(* IEC 61131-3 sources: AXOpen/src/template.axolibrary/ctrl/src/TemplateComponent, 1 file *)

(* ---- TemplateComponent.st ---- *)
USING AXOpen.Core;
USING AXOpen.Messaging;
USING AXOpen.Messaging.Static;
USING AXOpen.Components.Abstractions;
USING Siemens.Simatic.Hardware.Utilities;

NAMESPACE Template.Axolibrary
    {S7.extern=ReadWrite}
    CLASS TemplateComponent EXTENDS AXOpen.Core.AxoComponent
        VAR PUBLIC // HEADER
            {#ix-attr:[ReadOnly()]}
            Progress       :   INT;
        END_VAR

        VAR PUBLIC // TASKS
            {#ix-attr:[Container(Layout.Wrap)]}
            {#ix-attr:[ComponentDetails("Tasks")]}
            {#ix-set:AttributeName = "<#Restore#>"}
            RestoreTask : AXOpen.Core.AxoTask;
        END_VAR

        VAR PUBLIC // TEMPLATE TASKS
            {#ix-attr:[Container(Layout.Wrap)]}
            {#ix-attr:[ComponentDetails("Template tasks")]}
            {#ix-set:AttributeName = "<#TemplateTask_10steps_1#>"}
            TemplateTask_10steps_1 : AXOpen.Core.AxoTask;
            {#ix-attr:[Container(Layout.Wrap)]}
            {#ix-attr:[ComponentDetails("Template tasks")]}
            {#ix-set:AttributeName = "<#TemplateTask_10steps_2#>"}
            TemplateTask_10steps_2 : AXOpen.Core.AxoTask;
            {#ix-attr:[Container(Layout.Wrap)]}
            {#ix-attr:[ComponentDetails("Template tasks")]}
            {#ix-set:AttributeName = "<#TemplateTask_10steps_3#>"}
            TemplateTask_10steps_3 : AXOpen.Core.AxoTask;
            {#ix-attr:[Container(Layout.Wrap)]}
            {#ix-attr:[ComponentDetails("Template tasks")]}
            {#ix-set:AttributeName = "<#TemplateTask_10steps_4#>"}
            TemplateTask_10steps_4 : AXOpen.Core.AxoTask;
            {#ix-attr:[Container(Layout.Wrap)]}
            {#ix-attr:[ComponentDetails("Template tasks")]}
            {#ix-set:AttributeName = "<#TemplateTask_10steps_5#>"}
            TemplateTask_10steps_5 : AXOpen.Core.AxoTask;
            {#ix-attr:[Container(Layout.Wrap)]}
            {#ix-attr:[ComponentDetails("Template tasks")]}
            {#ix-set:AttributeName = "<#TemplateTask_10steps_6#>"}
            TemplateTask_10steps_6 : AXOpen.Core.AxoTask;

            {#ix-attr:[Container(Layout.Wrap)]}
            {#ix-attr:[ComponentDetails("Template tasks")]}
            {#ix-set:AttributeName = "<#TemplateTask_20steps_1#>"}
            TemplateTask_20steps_1 : AXOpen.Core.AxoTask;
            {#ix-attr:[Container(Layout.Wrap)]}
            {#ix-attr:[ComponentDetails("Template tasks")]}
            {#ix-set:AttributeName = "<#TemplateTask_20steps_2#>"}
            TemplateTask_20steps_2 : AXOpen.Core.AxoTask;
            {#ix-attr:[Container(Layout.Wrap)]}
            {#ix-attr:[ComponentDetails("Template tasks")]}
            {#ix-set:AttributeName = "<#TemplateTask_20steps_3#>"}
            TemplateTask_20steps_3 : AXOpen.Core.AxoTask;
            {#ix-attr:[Container(Layout.Wrap)]}
            {#ix-attr:[ComponentDetails("Template tasks")]}
            {#ix-set:AttributeName = "<#TemplateTask_20steps_4#>"}
            TemplateTask_20steps_4 : AXOpen.Core.AxoTask;
            {#ix-attr:[Container(Layout.Wrap)]}
            {#ix-attr:[ComponentDetails("Template tasks")]}
            {#ix-set:AttributeName = "<#TemplateTask_20steps_5#>"}
            TemplateTask_20steps_5 : AXOpen.Core.AxoTask;
            {#ix-attr:[Container(Layout.Wrap)]}
            {#ix-attr:[ComponentDetails("Template tasks")]}
            {#ix-set:AttributeName = "<#TemplateTask_20steps_6#>"}
            TemplateTask_20steps_6 : AXOpen.Core.AxoTask;

        END_VAR

        VAR PUBLIC // CONFIG
            {#ix-attr:[Container(Layout.Stack)]}
            {#ix-attr:[ComponentDetails("Config")]}
            {#ix-attr:[ReadOnly()]}
            Config  :   TemplateComponent_Config;
        END_VAR

        VAR PUBLIC // STATUS
            {#ix-attr:[Container(Layout.Stack)]}
            {#ix-attr:[ComponentDetails("Status")]}
            {#ix-attr:[ReadOnly()]}
            Status              :   TemplateComponent_Component_Status;
            Messenger           :   AXOpen.Messaging.Static.AxoMessenger;
            TaskMessenger       :   AXOpen.Messaging.Static.AxoMessenger;
        END_VAR

        VAR PUBLIC // HARDWARE SIGNALS
            {#ix-attr:[ComponentDetails("HARDWARE SIGNALS")]}
            {#ix-attr:[Container(Layout.Wrap)]}
            {#ix-attr:[Group(GroupLayout.GroupBox)]}
            {#ix-set:AttributeName = "<#Inputs#>"}
            {#ix-attr:[ReadOnly()]}
            Inputs              :  TemplateComponent_In;
            {#ix-attr:[ComponentDetails("HARDWARE SIGNALS")]}
            {#ix-attr:[Container(Layout.Wrap)]}
            {#ix-attr:[Group(GroupLayout.GroupBox)]}
            {#ix-set:AttributeName = "<#Outputs#>"}
            {#ix-attr:[ReadOnly()]}
            Outputs              :   TemplateComponent_Out;
        END_VAR

        VAR PUBLIC // HARDWARE DIAGNOSTICS TASK
            {#ix-attr:[Container(Layout.Stack)]}
            {#ix-attr:[ComponentDetails("Hardware diagnostics")]}
            {#ix-set:AttributeName = "<#Update diagnostics#>"}
            HardwareDiagnosticsTask :   AXOpen.Io.AxoHardwareDiagnostics;
        END_VAR

        VAR PRIVATE
            _progress       :   INT;
            _infoTimer      :   AXOpen.Timers.OnDelayTimer;
            _errorTimer     :   AXOpen.Timers.OnDelayTimer;
            _data_in        :   ARRAY[0..254] OF BYTE;
            _data_out_1     :   ARRAY[0..0] OF BYTE;
            _data_out_2     :   ARRAY[0..1] OF BYTE;
            _data_out_4     :   ARRAY[0..3] OF BYTE;
            _data_out_8     :   ARRAY[0..7] OF BYTE;
            _data_out_255   :   ARRAY[0..254] OF BYTE;
            _word           :   WORD;
            _dword          :   DWORD;

            _initHwCheckDone        :   BOOL;
            _retval                 :   WORD;
            _geoAddr                :   GeoAddr;
            _outHwid                :   UINT;
            _blink                  :   AXOpen.Timers.AxoBlinker;
            _inputsAddress          :   UDINT;
            _inputsCount            :   UINT;
            _outputsAddress         :   UDINT;
            _outputsCount           :   UINT;
        END_VAR

        ///<summary>
        /// Runs tasks and logic of this component.
        /// >[!IMPORTANT] This method must or one of its overloads be called cyclically.
        ///</summary>
        METHOD PUBLIC Run
            VAR_INPUT
                inParent    :   IAxoObject;
                hwID        :   UINT;
            END_VAR

            SUPER.Run(inParent);

            Messenger.Serve(THIS);

            Progress := _progress;

            IF NOT _initHwCheckDone THEN
                IF inParent = NULL THEN
                    Messenger.Activate(UINT#700, eAxoMessageCategory#ProgrammingError);
                    Status.Error.Id := UINT#700;
                    RETURN;
                END_IF;
                IF hwID = UINT#0 THEN
                    Messenger.Activate(UINT#701, eAxoMessageCategory#ProgrammingError);
                    Status.Error.Id := UINT#701;
                    RETURN;
                END_IF;

                Config.HWIDs.HW_Device := hwID;
                _retval := ReadSlotFromHardwareID(hardwareID := Config.HWIDs.HW_Device, geoAddr :=_geoAddr);
                IF _retval = WORD#8090 THEN
                    Messenger.Activate(UINT#702,eAxoMessageCategory#Error);
                    Status.Error.Id := UINT#702;
                    RETURN;
                END_IF;

                //******************Slot 1*****************//
                _geoAddr.Slot   :=  UINT#1;
                _geoAddr.HardwareType := UINT#4; // (4-Module)
                _retval := ReadHardwareIDFromSlot(geoAddr := _geoAddr, hardwareID => Config.HWIDs.HwID_in_1);
                IF Config.HWIDs.HwID_in_1 = UINT#0 THEN
                    Messenger.Activate(UINT#710,eAxoMessageCategory#Error);
                    Status.Error.Id := UINT#710;
                    RETURN;
                END_IF;
                IF _retval = WORD#8091 THEN
                    Messenger.Activate(UINT#711,eAxoMessageCategory#Error);
                    Status.Error.Id := UINT#711;
                    RETURN;
                END_IF;
                IF _retval = WORD#8094 THEN
                    Messenger.Activate(UINT#712,eAxoMessageCategory#Error);
                    Status.Error.Id := UINT#712;
                    RETURN;
                END_IF;
                IF _retval = WORD#8095 THEN
                    Messenger.Activate(UINT#713,eAxoMessageCategory#Error);
                    Status.Error.Id := UINT#713;
                    RETURN;
                END_IF;
                IF _retval = WORD#8096 THEN
                    Messenger.Activate(UINT#714,eAxoMessageCategory#Error);
                    Status.Error.Id := UINT#714;
                    RETURN;
                END_IF;
                IF _retval = WORD#8097 THEN
                    Messenger.Activate(UINT#715,eAxoMessageCategory#Error);
                    Status.Error.Id := UINT#715;
                    RETURN;
                END_IF;
                ReadHardwareIOAddress(hardwareID := (Config.HWIDs.HwID_in_1) , inputStartAddress => _inputsAddress , inputCount => _inputsCount , outputStartAddress => _outputsAddress , outputCount => _outputsCount);
                IF _inputsCount <> UINT#8 OR _outputsCount <> UINT#0 THEN
                    Messenger.Activate(UINT#716,eAxoMessageCategory#Error);
                    Status.Error.Id := UINT#716;
                    RETURN;
                END_IF;
                //******************Slot 2*****************//
                _geoAddr.Slot   :=  UINT#2;
                _geoAddr.HardwareType := UINT#4; // (4-Module)
                _retval := ReadHardwareIDFromSlot(geoAddr := _geoAddr, hardwareID => Config.HWIDs.HwID_in_2);
                IF Config.HWIDs.HwID_in_2 = UINT#0 THEN
                    Messenger.Activate(UINT#720,eAxoMessageCategory#Error);
                    Status.Error.Id := UINT#720;
                    RETURN;
                END_IF;
                IF _retval = WORD#8091 THEN
                    Messenger.Activate(UINT#721,eAxoMessageCategory#Error);
                    Status.Error.Id := UINT#721;
                    RETURN;
                END_IF;
                IF _retval = WORD#8094 THEN
                    Messenger.Activate(UINT#722,eAxoMessageCategory#Error);
                    Status.Error.Id := UINT#722;
                    RETURN;
                END_IF;
                IF _retval = WORD#8095 THEN
                    Messenger.Activate(UINT#723,eAxoMessageCategory#Error);
                    Status.Error.Id := UINT#723;
                    RETURN;
                END_IF;
                IF _retval = WORD#8096 THEN
                    Messenger.Activate(UINT#724,eAxoMessageCategory#Error);
                    Status.Error.Id := UINT#724;
                    RETURN;
                END_IF;
                IF _retval = WORD#8097 THEN
                    Messenger.Activate(UINT#725,eAxoMessageCategory#Error);
                    Status.Error.Id := UINT#725;
                    RETURN;
                END_IF;
                ReadHardwareIOAddress(hardwareID := (Config.HWIDs.HwID_in_2) , inputStartAddress => _inputsAddress , inputCount => _inputsCount , outputStartAddress => _outputsAddress , outputCount => _outputsCount);
                IF _inputsCount <> UINT#8 OR _outputsCount <> UINT#0 THEN
                    Messenger.Activate(UINT#726,eAxoMessageCategory#Error);
                    Status.Error.Id := UINT#726;
                    RETURN;
                END_IF;
                //******************Slot 3*****************//
                _geoAddr.Slot   :=  UINT#3;
                _geoAddr.HardwareType := UINT#4; // (4-Module)
                _retval := ReadHardwareIDFromSlot(geoAddr := _geoAddr, hardwareID => Config.HWIDs.HwID_in_3);
                IF Config.HWIDs.HwID_in_1 = UINT#0 THEN
                    Messenger.Activate(UINT#730,eAxoMessageCategory#Error);
                    Status.Error.Id := UINT#730;
                    RETURN;
                END_IF;
                IF _retval = WORD#8091 THEN
                    Messenger.Activate(UINT#731,eAxoMessageCategory#Error);
                    Status.Error.Id := UINT#731;
                    RETURN;
                END_IF;
                IF _retval = WORD#8094 THEN
                    Messenger.Activate(UINT#732,eAxoMessageCategory#Error);
                    Status.Error.Id := UINT#732;
                    RETURN;
                END_IF;
                IF _retval = WORD#8095 THEN
                    Messenger.Activate(UINT#733,eAxoMessageCategory#Error);
                    Status.Error.Id := UINT#733;
                    RETURN;
                END_IF;
                IF _retval = WORD#8096 THEN
                    Messenger.Activate(UINT#734,eAxoMessageCategory#Error);
                    Status.Error.Id := UINT#734;
                    RETURN;
                END_IF;
                IF _retval = WORD#8097 THEN
                    Messenger.Activate(UINT#735,eAxoMessageCategory#Error);
                    Status.Error.Id := UINT#735;
                    RETURN;
                END_IF;
                ReadHardwareIOAddress(hardwareID := (Config.HWIDs.HwID_in_3) , inputStartAddress => _inputsAddress , inputCount => _inputsCount , outputStartAddress => _outputsAddress , outputCount => _outputsCount);
                IF _inputsCount <> UINT#8 OR _outputsCount <> UINT#0 THEN
                    Messenger.Activate(UINT#736,eAxoMessageCategory#Error);
                    Status.Error.Id := UINT#736;
                    RETURN;
                END_IF;
                //******************Slot 4*****************//
                _geoAddr.Slot   :=  UINT#4;
                _geoAddr.HardwareType := UINT#4; // (4-Module)
                _retval := ReadHardwareIDFromSlot(geoAddr := _geoAddr, hardwareID => Config.HWIDs.HwID_in_4);
                IF Config.HWIDs.HwID_in_4 = UINT#0 THEN
                    Messenger.Activate(UINT#740,eAxoMessageCategory#Error);
                    Status.Error.Id := UINT#740;
                    RETURN;
                END_IF;
                IF _retval = WORD#8091 THEN
                    Messenger.Activate(UINT#741,eAxoMessageCategory#Error);
                    Status.Error.Id := UINT#741;
                    RETURN;
                END_IF;
                IF _retval = WORD#8094 THEN
                    Messenger.Activate(UINT#742,eAxoMessageCategory#Error);
                    Status.Error.Id := UINT#742;
                    RETURN;
                END_IF;
                IF _retval = WORD#8095 THEN
                    Messenger.Activate(UINT#743,eAxoMessageCategory#Error);
                    Status.Error.Id := UINT#743;
                    RETURN;
                END_IF;
                IF _retval = WORD#8096 THEN
                    Messenger.Activate(UINT#744,eAxoMessageCategory#Error);
                    Status.Error.Id := UINT#744;
                    RETURN;
                END_IF;
                IF _retval = WORD#8097 THEN
                    Messenger.Activate(UINT#745,eAxoMessageCategory#Error);
                    Status.Error.Id := UINT#745;
                    RETURN;
                END_IF;
                ReadHardwareIOAddress(hardwareID := (Config.HWIDs.HwID_in_4) , inputStartAddress => _inputsAddress , inputCount => _inputsCount , outputStartAddress => _outputsAddress , outputCount => _outputsCount);
                IF _inputsCount <> UINT#8 OR _outputsCount <> UINT#0 THEN
                    Messenger.Activate(UINT#746,eAxoMessageCategory#Error);
                    Status.Error.Id := UINT#746;
                    RETURN;
                END_IF;
                //******************Slot 5*****************//
                _geoAddr.Slot   :=  UINT#5;
                _geoAddr.HardwareType := UINT#4; // (4-Module)
                _retval := ReadHardwareIDFromSlot(geoAddr := _geoAddr, hardwareID => Config.HWIDs.HwID_in_5);
                IF Config.HWIDs.HwID_in_5 = UINT#0 THEN
                    Messenger.Activate(UINT#750,eAxoMessageCategory#Error);
                    Status.Error.Id := UINT#750;
                    RETURN;
                END_IF;
                IF _retval = WORD#8091 THEN
                    Messenger.Activate(UINT#751,eAxoMessageCategory#Error);
                    Status.Error.Id := UINT#751;
                    RETURN;
                END_IF;
                IF _retval = WORD#8094 THEN
                    Messenger.Activate(UINT#752,eAxoMessageCategory#Error);
                    Status.Error.Id := UINT#752;
                    RETURN;
                END_IF;
                IF _retval = WORD#8095 THEN
                    Messenger.Activate(UINT#753,eAxoMessageCategory#Error);
                    Status.Error.Id := UINT#753;
                    RETURN;
                END_IF;
                IF _retval = WORD#8096 THEN
                    Messenger.Activate(UINT#754,eAxoMessageCategory#Error);
                    Status.Error.Id := UINT#754;
                    RETURN;
                END_IF;
                IF _retval = WORD#8097 THEN
                    Messenger.Activate(UINT#755,eAxoMessageCategory#Error);
                    Status.Error.Id := UINT#755;
                    RETURN;
                END_IF;
                ReadHardwareIOAddress(hardwareID := (Config.HWIDs.HwID_in_5) , inputStartAddress => _inputsAddress , inputCount => _inputsCount , outputStartAddress => _outputsAddress , outputCount => _outputsCount);
                IF _inputsCount <> UINT#8 OR _outputsCount <> UINT#0 THEN
                    Messenger.Activate(UINT#756,eAxoMessageCategory#Error);
                    Status.Error.Id := UINT#756;
                    RETURN;
                END_IF;
                //******************Slot 6*****************//
                _geoAddr.Slot   :=  UINT#6;
                _geoAddr.HardwareType := UINT#4; // (4-Module)
                _retval := ReadHardwareIDFromSlot(geoAddr := _geoAddr, hardwareID => Config.HWIDs.HwID_in_6);
                IF Config.HWIDs.HwID_in_6 = UINT#0 THEN
                    Messenger.Activate(UINT#760,eAxoMessageCategory#Error);
                    Status.Error.Id := UINT#760;
                    RETURN;
                END_IF;
                IF _retval = WORD#8091 THEN
                    Messenger.Activate(UINT#761,eAxoMessageCategory#Error);
                    Status.Error.Id := UINT#761;
                    RETURN;
                END_IF;
                IF _retval = WORD#8094 THEN
                    Messenger.Activate(UINT#762,eAxoMessageCategory#Error);
                    Status.Error.Id := UINT#762;
                    RETURN;
                END_IF;
                IF _retval = WORD#8095 THEN
                    Messenger.Activate(UINT#763,eAxoMessageCategory#Error);
                    Status.Error.Id := UINT#763;
                    RETURN;
                END_IF;
                IF _retval = WORD#8096 THEN
                    Messenger.Activate(UINT#764,eAxoMessageCategory#Error);
                    Status.Error.Id := UINT#764;
                    RETURN;
                END_IF;
                IF _retval = WORD#8097 THEN
                    Messenger.Activate(UINT#765,eAxoMessageCategory#Error);
                    Status.Error.Id := UINT#765;
                    RETURN;
                END_IF;
                ReadHardwareIOAddress(hardwareID := (Config.HWIDs.HwID_in_6) , inputStartAddress => _inputsAddress , inputCount => _inputsCount , outputStartAddress => _outputsAddress , outputCount => _outputsCount);
                IF _inputsCount <> UINT#8 OR _outputsCount <> UINT#0 THEN
                    Messenger.Activate(UINT#766,eAxoMessageCategory#Error);
                    Status.Error.Id := UINT#766;
                    RETURN;
                END_IF;
                //******************Slot 7*****************//
                _geoAddr.Slot   :=  UINT#7;
                _geoAddr.HardwareType := UINT#4; // (4-Module)
                _retval := ReadHardwareIDFromSlot(geoAddr := _geoAddr, hardwareID => Config.HWIDs.HwID_in_7);
                IF Config.HWIDs.HwID_in_7 = UINT#0 THEN
                    Messenger.Activate(UINT#770,eAxoMessageCategory#Error);
                    Status.Error.Id := UINT#770;
                    RETURN;
                END_IF;
                IF _retval = WORD#8091 THEN
                    Messenger.Activate(UINT#771,eAxoMessageCategory#Error);
                    Status.Error.Id := UINT#771;
                    RETURN;
                END_IF;
                IF _retval = WORD#8094 THEN
                    Messenger.Activate(UINT#772,eAxoMessageCategory#Error);
                    Status.Error.Id := UINT#772;
                    RETURN;
                END_IF;
                IF _retval = WORD#8095 THEN
                    Messenger.Activate(UINT#773,eAxoMessageCategory#Error);
                    Status.Error.Id := UINT#773;
                    RETURN;
                END_IF;
                IF _retval = WORD#8096 THEN
                    Messenger.Activate(UINT#774,eAxoMessageCategory#Error);
                    Status.Error.Id := UINT#774;
                    RETURN;
                END_IF;
                IF _retval = WORD#8097 THEN
                    Messenger.Activate(UINT#775,eAxoMessageCategory#Error);
                    Status.Error.Id := UINT#775;
                    RETURN;
                END_IF;
                ReadHardwareIOAddress(hardwareID := (Config.HWIDs.HwID_in_7) , inputStartAddress => _inputsAddress , inputCount => _inputsCount , outputStartAddress => _outputsAddress , outputCount => _outputsCount);
                IF _inputsCount <> UINT#8 OR _outputsCount <> UINT#0 THEN
                    Messenger.Activate(UINT#776,eAxoMessageCategory#Error);
                    Status.Error.Id := UINT#776;
                    RETURN;
                END_IF;
                //******************Slot 8*****************//
                _geoAddr.Slot   :=  UINT#8;
                _geoAddr.HardwareType := UINT#4; // (4-Module)
                _retval := ReadHardwareIDFromSlot(geoAddr := _geoAddr, hardwareID => Config.HWIDs.HwID_in_8);
                IF Config.HWIDs.HwID_in_8 = UINT#0 THEN
                    Messenger.Activate(UINT#780,eAxoMessageCategory#Error);
                    Status.Error.Id := UINT#780;
                    RETURN;
                END_IF;
                IF _retval = WORD#8091 THEN
                    Messenger.Activate(UINT#781,eAxoMessageCategory#Error);
                    Status.Error.Id := UINT#781;
                    RETURN;
                END_IF;
                IF _retval = WORD#8094 THEN
                    Messenger.Activate(UINT#782,eAxoMessageCategory#Error);
                    Status.Error.Id := UINT#782;
                    RETURN;
                END_IF;
                IF _retval = WORD#8095 THEN
                    Messenger.Activate(UINT#783,eAxoMessageCategory#Error);
                    Status.Error.Id := UINT#783;
                    RETURN;
                END_IF;
                IF _retval = WORD#8096 THEN
                    Messenger.Activate(UINT#784,eAxoMessageCategory#Error);
                    Status.Error.Id := UINT#784;
                    RETURN;
                END_IF;
                IF _retval = WORD#8097 THEN
                    Messenger.Activate(UINT#785,eAxoMessageCategory#Error);
                    Status.Error.Id := UINT#785;
                    RETURN;
                END_IF;
                ReadHardwareIOAddress(hardwareID := (Config.HWIDs.HwID_in_8) , inputStartAddress => _inputsAddress , inputCount => _inputsCount , outputStartAddress => _outputsAddress , outputCount => _outputsCount);
                IF _inputsCount <> UINT#8 OR _outputsCount <> UINT#0 THEN
                    Messenger.Activate(UINT#786,eAxoMessageCategory#Error);
                    Status.Error.Id := UINT#786;
                    RETURN;
                END_IF;
                //******************Slot 9*****************//
                _geoAddr.Slot   :=  UINT#9;
                _geoAddr.HardwareType := UINT#4; // (4-Module)
                _retval := ReadHardwareIDFromSlot(geoAddr := _geoAddr, hardwareID => Config.HWIDs.HwID_in_9);
                IF Config.HWIDs.HwID_in_9 = UINT#0 THEN
                    Messenger.Activate(UINT#790,eAxoMessageCategory#Error);
                    Status.Error.Id := UINT#790;
                    RETURN;
                END_IF;
                IF _retval = WORD#8091 THEN
                    Messenger.Activate(UINT#791,eAxoMessageCategory#Error);
                    Status.Error.Id := UINT#791;
                    RETURN;
                END_IF;
                IF _retval = WORD#8094 THEN
                    Messenger.Activate(UINT#792,eAxoMessageCategory#Error);
                    Status.Error.Id := UINT#792;
                    RETURN;
                END_IF;
                IF _retval = WORD#8095 THEN
                    Messenger.Activate(UINT#793,eAxoMessageCategory#Error);
                    Status.Error.Id := UINT#793;
                    RETURN;
                END_IF;
                IF _retval = WORD#8096 THEN
                    Messenger.Activate(UINT#794,eAxoMessageCategory#Error);
                    Status.Error.Id := UINT#794;
                    RETURN;
                END_IF;
                IF _retval = WORD#8097 THEN
                    Messenger.Activate(UINT#795,eAxoMessageCategory#Error);
                    Status.Error.Id := UINT#795;
                    RETURN;
                END_IF;
                ReadHardwareIOAddress(hardwareID := (Config.HWIDs.HwID_in_9) , inputStartAddress => _inputsAddress , inputCount => _inputsCount , outputStartAddress => _outputsAddress , outputCount => _outputsCount);
                IF _inputsCount <> UINT#8 OR _outputsCount <> UINT#0 THEN
                    Messenger.Activate(UINT#796,eAxoMessageCategory#Error);
                    Status.Error.Id := UINT#796;
                    RETURN;
                END_IF;
                //******************Slot 10*****************//
                _geoAddr.Slot   :=  UINT#10;
                _geoAddr.HardwareType := UINT#4; // (4-Module)
                _retval := ReadHardwareIDFromSlot(geoAddr := _geoAddr, hardwareID => Config.HWIDs.HwID_in_10);
                IF Config.HWIDs.HwID_in_10 = UINT#0 THEN
                    Messenger.Activate(UINT#800,eAxoMessageCategory#Error);
                    Status.Error.Id := UINT#800;
                    RETURN;
                END_IF;
                IF _retval = WORD#8091 THEN
                    Messenger.Activate(UINT#801,eAxoMessageCategory#Error);
                    Status.Error.Id := UINT#801;
                    RETURN;
                END_IF;
                IF _retval = WORD#8094 THEN
                    Messenger.Activate(UINT#802,eAxoMessageCategory#Error);
                    Status.Error.Id := UINT#802;
                    RETURN;
                END_IF;
                IF _retval = WORD#8095 THEN
                    Messenger.Activate(UINT#803,eAxoMessageCategory#Error);
                    Status.Error.Id := UINT#803;
                    RETURN;
                END_IF;
                IF _retval = WORD#8096 THEN
                    Messenger.Activate(UINT#804,eAxoMessageCategory#Error);
                    Status.Error.Id := UINT#804;
                    RETURN;
                END_IF;
                IF _retval = WORD#8097 THEN
                    Messenger.Activate(UINT#805,eAxoMessageCategory#Error);
                    Status.Error.Id := UINT#805;
                    RETURN;
                END_IF;
                ReadHardwareIOAddress(hardwareID := (Config.HWIDs.HwID_in_10) , inputStartAddress => _inputsAddress , inputCount => _inputsCount , outputStartAddress => _outputsAddress , outputCount => _outputsCount);
                IF _inputsCount <> UINT#8 OR _outputsCount <> UINT#0 THEN
                    Messenger.Activate(UINT#806,eAxoMessageCategory#Error);
                    Status.Error.Id := UINT#806;
                    RETURN;
                END_IF;
                //******************Slot 11*****************//
                _geoAddr.Slot   :=  UINT#11;
                _geoAddr.HardwareType := UINT#4; // (4-Module)
                _retval := ReadHardwareIDFromSlot(geoAddr := _geoAddr, hardwareID => Config.HWIDs.HwID_in_11);
                IF Config.HWIDs.HwID_in_11 = UINT#0 THEN
                    Messenger.Activate(UINT#810,eAxoMessageCategory#Error);
                    Status.Error.Id := UINT#810;
                    RETURN;
                END_IF;
                IF _retval = WORD#8091 THEN
                    Messenger.Activate(UINT#811,eAxoMessageCategory#Error);
                    Status.Error.Id := UINT#811;
                    RETURN;
                END_IF;
                IF _retval = WORD#8094 THEN
                    Messenger.Activate(UINT#812,eAxoMessageCategory#Error);
                    Status.Error.Id := UINT#812;
                    RETURN;
                END_IF;
                IF _retval = WORD#8095 THEN
                    Messenger.Activate(UINT#813,eAxoMessageCategory#Error);
                    Status.Error.Id := UINT#813;
                    RETURN;
                END_IF;
                IF _retval = WORD#8096 THEN
                    Messenger.Activate(UINT#814,eAxoMessageCategory#Error);
                    Status.Error.Id := UINT#814;
                    RETURN;
                END_IF;
                IF _retval = WORD#8097 THEN
                    Messenger.Activate(UINT#815,eAxoMessageCategory#Error);
                    Status.Error.Id := UINT#815;
                    RETURN;
                END_IF;
                ReadHardwareIOAddress(hardwareID := (Config.HWIDs.HwID_in_11) , inputStartAddress => _inputsAddress , inputCount => _inputsCount , outputStartAddress => _outputsAddress , outputCount => _outputsCount);
                IF _inputsCount <> UINT#8 OR _outputsCount <> UINT#0 THEN
                    Messenger.Activate(UINT#816,eAxoMessageCategory#Error);
                    Status.Error.Id := UINT#816;
                    RETURN;
                END_IF;
                //******************Slot 12*****************//
                _geoAddr.Slot   :=  UINT#12;
                _geoAddr.HardwareType := UINT#4; // (4-Module)
                _retval := ReadHardwareIDFromSlot(geoAddr := _geoAddr, hardwareID => Config.HWIDs.HwID_in_12);
                IF Config.HWIDs.HwID_in_12 = UINT#0 THEN
                    Messenger.Activate(UINT#820,eAxoMessageCategory#Error);
                    Status.Error.Id := UINT#820;
                    RETURN;
                END_IF;
                IF _retval = WORD#8091 THEN
                    Messenger.Activate(UINT#821,eAxoMessageCategory#Error);
                    Status.Error.Id := UINT#821;
                    RETURN;
                END_IF;
                IF _retval = WORD#8094 THEN
                    Messenger.Activate(UINT#822,eAxoMessageCategory#Error);
                    Status.Error.Id := UINT#822;
                    RETURN;
                END_IF;
                IF _retval = WORD#8095 THEN
                    Messenger.Activate(UINT#823,eAxoMessageCategory#Error);
                    Status.Error.Id := UINT#823;
                    RETURN;
                END_IF;
                IF _retval = WORD#8096 THEN
                    Messenger.Activate(UINT#824,eAxoMessageCategory#Error);
                    Status.Error.Id := UINT#824;
                    RETURN;
                END_IF;
                IF _retval = WORD#8097 THEN
                    Messenger.Activate(UINT#825,eAxoMessageCategory#Error);
                    Status.Error.Id := UINT#825;
                    RETURN;
                END_IF;
                ReadHardwareIOAddress(hardwareID := (Config.HWIDs.HwID_in_12) , inputStartAddress => _inputsAddress , inputCount => _inputsCount , outputStartAddress => _outputsAddress , outputCount => _outputsCount);
                IF _inputsCount <> UINT#8 OR _outputsCount <> UINT#0 THEN
                    Messenger.Activate(UINT#826,eAxoMessageCategory#Error);
                    Status.Error.Id := UINT#826;
                    RETURN;
                END_IF;
                //******************Slot 13*****************//
                _geoAddr.Slot   :=  UINT#13;
                _geoAddr.HardwareType := UINT#4; // (4-Module)
                _retval := ReadHardwareIDFromSlot(geoAddr := _geoAddr, hardwareID => Config.HWIDs.HwID_in_13);
                IF Config.HWIDs.HwID_in_13 = UINT#0 THEN
                    Messenger.Activate(UINT#830,eAxoMessageCategory#Error);
                    Status.Error.Id := UINT#830;
                    RETURN;
                END_IF;
                IF _retval = WORD#8091 THEN
                    Messenger.Activate(UINT#831,eAxoMessageCategory#Error);
                    Status.Error.Id := UINT#831;
                    RETURN;
                END_IF;
                IF _retval = WORD#8094 THEN
                    Messenger.Activate(UINT#832,eAxoMessageCategory#Error);
                    Status.Error.Id := UINT#832;
                    RETURN;
                END_IF;
                IF _retval = WORD#8095 THEN
                    Messenger.Activate(UINT#833,eAxoMessageCategory#Error);
                    Status.Error.Id := UINT#833;
                    RETURN;
                END_IF;
                IF _retval = WORD#8096 THEN
                    Messenger.Activate(UINT#834,eAxoMessageCategory#Error);
                    Status.Error.Id := UINT#834;
                    RETURN;
                END_IF;
                IF _retval = WORD#8097 THEN
                    Messenger.Activate(UINT#835,eAxoMessageCategory#Error);
                    Status.Error.Id := UINT#835;
                    RETURN;
                END_IF;
                ReadHardwareIOAddress(hardwareID := (Config.HWIDs.HwID_in_13) , inputStartAddress => _inputsAddress , inputCount => _inputsCount , outputStartAddress => _outputsAddress , outputCount => _outputsCount);
                IF _inputsCount <> UINT#8 OR _outputsCount <> UINT#0 THEN
                    Messenger.Activate(UINT#836,eAxoMessageCategory#Error);
                    Status.Error.Id := UINT#836;
                    RETURN;
                END_IF;
                //******************Slot 14*****************//
                _geoAddr.Slot   :=  UINT#14;
                _geoAddr.HardwareType := UINT#4; // (4-Module)
                _retval := ReadHardwareIDFromSlot(geoAddr := _geoAddr, hardwareID => Config.HWIDs.HwID_in_14);
                IF Config.HWIDs.HwID_in_14 = UINT#0 THEN
                    Messenger.Activate(UINT#840,eAxoMessageCategory#Error);
                    Status.Error.Id := UINT#840;
                    RETURN;
                END_IF;
                IF _retval = WORD#8091 THEN
                    Messenger.Activate(UINT#841,eAxoMessageCategory#Error);
                    Status.Error.Id := UINT#841;
                    RETURN;
                END_IF;
                IF _retval = WORD#8094 THEN
                    Messenger.Activate(UINT#842,eAxoMessageCategory#Error);
                    Status.Error.Id := UINT#842;
                    RETURN;
                END_IF;
                IF _retval = WORD#8095 THEN
                    Messenger.Activate(UINT#843,eAxoMessageCategory#Error);
                    Status.Error.Id := UINT#843;
                    RETURN;
                END_IF;
                IF _retval = WORD#8096 THEN
                    Messenger.Activate(UINT#844,eAxoMessageCategory#Error);
                    Status.Error.Id := UINT#844;
                    RETURN;
                END_IF;
                IF _retval = WORD#8097 THEN
                    Messenger.Activate(UINT#845,eAxoMessageCategory#Error);
                    Status.Error.Id := UINT#845;
                    RETURN;
                END_IF;
                ReadHardwareIOAddress(hardwareID := (Config.HWIDs.HwID_in_14) , inputStartAddress => _inputsAddress , inputCount => _inputsCount , outputStartAddress => _outputsAddress , outputCount => _outputsCount);
                IF _inputsCount <> UINT#8 OR _outputsCount <> UINT#0 THEN
                    Messenger.Activate(UINT#846,eAxoMessageCategory#Error);
                    Status.Error.Id := UINT#846;
                    RETURN;
                END_IF;
                //******************Slot 15*****************//
                _geoAddr.Slot   :=  UINT#15;
                _geoAddr.HardwareType := UINT#4; // (4-Module)
                _retval := ReadHardwareIDFromSlot(geoAddr := _geoAddr, hardwareID => Config.HWIDs.HwID_in_15);
                IF Config.HWIDs.HwID_in_15 = UINT#0 THEN
                    Messenger.Activate(UINT#850,eAxoMessageCategory#Error);
                    Status.Error.Id := UINT#850;
                    RETURN;
                END_IF;
                IF _retval = WORD#8091 THEN
                    Messenger.Activate(UINT#851,eAxoMessageCategory#Error);
                    Status.Error.Id := UINT#851;
                    RETURN;
                END_IF;
                IF _retval = WORD#8094 THEN
                    Messenger.Activate(UINT#852,eAxoMessageCategory#Error);
                    Status.Error.Id := UINT#852;
                    RETURN;
                END_IF;
                IF _retval = WORD#8095 THEN
                    Messenger.Activate(UINT#853,eAxoMessageCategory#Error);
                    Status.Error.Id := UINT#853;
                    RETURN;
                END_IF;
                IF _retval = WORD#8096 THEN
                    Messenger.Activate(UINT#854,eAxoMessageCategory#Error);
                    Status.Error.Id := UINT#854;
                    RETURN;
                END_IF;
                IF _retval = WORD#8097 THEN
                    Messenger.Activate(UINT#855,eAxoMessageCategory#Error);
                    Status.Error.Id := UINT#855;
                    RETURN;
                END_IF;
                ReadHardwareIOAddress(hardwareID := (Config.HWIDs.HwID_in_15) , inputStartAddress => _inputsAddress , inputCount => _inputsCount , outputStartAddress => _outputsAddress , outputCount => _outputsCount);
                IF _inputsCount <> UINT#8 OR _outputsCount <> UINT#0 THEN
                    Messenger.Activate(UINT#856,eAxoMessageCategory#Error);
                    Status.Error.Id := UINT#856;
                    RETURN;
                END_IF;
                //******************Slot 16*****************//
                _geoAddr.Slot   :=  UINT#16;
                _geoAddr.HardwareType := UINT#4; // (4-Module)
                _retval := ReadHardwareIDFromSlot(geoAddr := _geoAddr, hardwareID => Config.HWIDs.HwID_in_16);
                IF Config.HWIDs.HwID_in_16 = UINT#0 THEN
                    Messenger.Activate(UINT#860,eAxoMessageCategory#Error);
                    Status.Error.Id := UINT#860;
                    RETURN;
                END_IF;
                IF _retval = WORD#8091 THEN
                    Messenger.Activate(UINT#861,eAxoMessageCategory#Error);
                    Status.Error.Id := UINT#861;
                    RETURN;
                END_IF;
                IF _retval = WORD#8094 THEN
                    Messenger.Activate(UINT#862,eAxoMessageCategory#Error);
                    Status.Error.Id := UINT#862;
                    RETURN;
                END_IF;
                IF _retval = WORD#8095 THEN
                    Messenger.Activate(UINT#863,eAxoMessageCategory#Error);
                    Status.Error.Id := UINT#863;
                    RETURN;
                END_IF;
                IF _retval = WORD#8096 THEN
                    Messenger.Activate(UINT#864,eAxoMessageCategory#Error);
                    Status.Error.Id := UINT#864;
                    RETURN;
                END_IF;
                IF _retval = WORD#8097 THEN
                    Messenger.Activate(UINT#865,eAxoMessageCategory#Error);
                    Status.Error.Id := UINT#865;
                    RETURN;
                END_IF;
                ReadHardwareIOAddress(hardwareID := (Config.HWIDs.HwID_in_16) , inputStartAddress => _inputsAddress , inputCount => _inputsCount , outputStartAddress => _outputsAddress , outputCount => _outputsCount);
                IF _inputsCount <> UINT#8 OR _outputsCount <> UINT#0 THEN
                    Messenger.Activate(UINT#866,eAxoMessageCategory#Error);
                    Status.Error.Id := UINT#866;
                    RETURN;
                END_IF;
                //******************Slot 17*****************//
                _geoAddr.Slot   :=  UINT#17;
                _geoAddr.HardwareType := UINT#4; // (4-Module)
                _retval := ReadHardwareIDFromSlot(geoAddr := _geoAddr, hardwareID => Config.HWIDs.HwID_in_17);
                IF Config.HWIDs.HwID_in_17 = UINT#0 THEN
                    Messenger.Activate(UINT#870,eAxoMessageCategory#Error);
                    Status.Error.Id := UINT#870;
                    RETURN;
                END_IF;
                IF _retval = WORD#8091 THEN
                    Messenger.Activate(UINT#871,eAxoMessageCategory#Error);
                    Status.Error.Id := UINT#871;
                    RETURN;
                END_IF;
                IF _retval = WORD#8094 THEN
                    Messenger.Activate(UINT#872,eAxoMessageCategory#Error);
                    Status.Error.Id := UINT#872;
                    RETURN;
                END_IF;
                IF _retval = WORD#8095 THEN
                    Messenger.Activate(UINT#873,eAxoMessageCategory#Error);
                    Status.Error.Id := UINT#873;
                    RETURN;
                END_IF;
                IF _retval = WORD#8096 THEN
                    Messenger.Activate(UINT#874,eAxoMessageCategory#Error);
                    Status.Error.Id := UINT#874;
                    RETURN;
                END_IF;
                IF _retval = WORD#8097 THEN
                    Messenger.Activate(UINT#875,eAxoMessageCategory#Error);
                    Status.Error.Id := UINT#875;
                    RETURN;
                END_IF;
                ReadHardwareIOAddress(hardwareID := (Config.HWIDs.HwID_in_17) , inputStartAddress => _inputsAddress , inputCount => _inputsCount , outputStartAddress => _outputsAddress , outputCount => _outputsCount);
                IF _inputsCount <> UINT#8 OR _outputsCount <> UINT#0 THEN
                    Messenger.Activate(UINT#876,eAxoMessageCategory#Error);
                    Status.Error.Id := UINT#876;
                    RETURN;
                END_IF;
                //******************Slot 18*****************//
                _geoAddr.Slot   :=  UINT#18;
                _geoAddr.HardwareType := UINT#4; // (4-Module)
                _retval := ReadHardwareIDFromSlot(geoAddr := _geoAddr, hardwareID => Config.HWIDs.HwID_in_18);
                IF Config.HWIDs.HwID_in_18 = UINT#0 THEN
                    Messenger.Activate(UINT#880,eAxoMessageCategory#Error);
                    Status.Error.Id := UINT#880;
                    RETURN;
                END_IF;
                IF _retval = WORD#8091 THEN
                    Messenger.Activate(UINT#881,eAxoMessageCategory#Error);
                    Status.Error.Id := UINT#881;
                    RETURN;
                END_IF;
                IF _retval = WORD#8094 THEN
                    Messenger.Activate(UINT#882,eAxoMessageCategory#Error);
                    Status.Error.Id := UINT#882;
                    RETURN;
                END_IF;
                IF _retval = WORD#8095 THEN
                    Messenger.Activate(UINT#883,eAxoMessageCategory#Error);
                    Status.Error.Id := UINT#883;
                    RETURN;
                END_IF;
                IF _retval = WORD#8096 THEN
                    Messenger.Activate(UINT#884,eAxoMessageCategory#Error);
                    Status.Error.Id := UINT#884;
                    RETURN;
                END_IF;
                IF _retval = WORD#8097 THEN
                    Messenger.Activate(UINT#885,eAxoMessageCategory#Error);
                    Status.Error.Id := UINT#885;
                    RETURN;
                END_IF;
                ReadHardwareIOAddress(hardwareID := (Config.HWIDs.HwID_in_18) , inputStartAddress => _inputsAddress , inputCount => _inputsCount , outputStartAddress => _outputsAddress , outputCount => _outputsCount);
                IF _inputsCount <> UINT#8 OR _outputsCount <> UINT#0 THEN
                    Messenger.Activate(UINT#886,eAxoMessageCategory#Error);
                    Status.Error.Id := UINT#886;
                    RETURN;
                END_IF;
                //******************Slot 19*****************//
                _geoAddr.Slot   :=  UINT#19;
                _geoAddr.HardwareType := UINT#4; // (4-Module)
                _retval := ReadHardwareIDFromSlot(geoAddr := _geoAddr, hardwareID => Config.HWIDs.HwID_in_19);
                IF Config.HWIDs.HwID_in_19 = UINT#0 THEN
                    Messenger.Activate(UINT#890,eAxoMessageCategory#Error);
                    Status.Error.Id := UINT#890;
                    RETURN;
                END_IF;
                IF _retval = WORD#8091 THEN
                    Messenger.Activate(UINT#891,eAxoMessageCategory#Error);
                    Status.Error.Id := UINT#891;
                    RETURN;
                END_IF;
                IF _retval = WORD#8094 THEN
                    Messenger.Activate(UINT#892,eAxoMessageCategory#Error);
                    Status.Error.Id := UINT#892;
                    RETURN;
                END_IF;
                IF _retval = WORD#8095 THEN
                    Messenger.Activate(UINT#893,eAxoMessageCategory#Error);
                    Status.Error.Id := UINT#893;
                    RETURN;
                END_IF;
                IF _retval = WORD#8096 THEN
                    Messenger.Activate(UINT#894,eAxoMessageCategory#Error);
                    Status.Error.Id := UINT#894;
                    RETURN;
                END_IF;
                IF _retval = WORD#8097 THEN
                    Messenger.Activate(UINT#895,eAxoMessageCategory#Error);
                    Status.Error.Id := UINT#895;
                    RETURN;
                END_IF;
                ReadHardwareIOAddress(hardwareID := (Config.HWIDs.HwID_in_19) , inputStartAddress => _inputsAddress , inputCount => _inputsCount , outputStartAddress => _outputsAddress , outputCount => _outputsCount);
                IF _inputsCount <> UINT#8 OR _outputsCount <> UINT#0 THEN
                    Messenger.Activate(UINT#896,eAxoMessageCategory#Error);
                    Status.Error.Id := UINT#896;
                    RETURN;
                END_IF;
                //******************Slot 20*****************//
                _geoAddr.Slot   :=  UINT#20;
                _geoAddr.HardwareType := UINT#4; // (4-Module)
                _retval := ReadHardwareIDFromSlot(geoAddr := _geoAddr, hardwareID => Config.HWIDs.HwID_in_20);
                IF Config.HWIDs.HwID_in_20 = UINT#0 THEN
                    Messenger.Activate(UINT#900,eAxoMessageCategory#Error);
                    Status.Error.Id := UINT#900;
                    RETURN;
                END_IF;
                IF _retval = WORD#8091 THEN
                    Messenger.Activate(UINT#901,eAxoMessageCategory#Error);
                    Status.Error.Id := UINT#901;
                    RETURN;
                END_IF;
                IF _retval = WORD#8094 THEN
                    Messenger.Activate(UINT#902,eAxoMessageCategory#Error);
                    Status.Error.Id := UINT#902;
                    RETURN;
                END_IF;
                IF _retval = WORD#8095 THEN
                    Messenger.Activate(UINT#903,eAxoMessageCategory#Error);
                    Status.Error.Id := UINT#903;
                    RETURN;
                END_IF;
                IF _retval = WORD#8096 THEN
                    Messenger.Activate(UINT#904,eAxoMessageCategory#Error);
                    Status.Error.Id := UINT#904;
                    RETURN;
                END_IF;
                IF _retval = WORD#8097 THEN
                    Messenger.Activate(UINT#905,eAxoMessageCategory#Error);
                    Status.Error.Id := UINT#905;
                    RETURN;
                END_IF;
                ReadHardwareIOAddress(hardwareID := (Config.HWIDs.HwID_in_20) , inputStartAddress => _inputsAddress , inputCount => _inputsCount , outputStartAddress => _outputsAddress , outputCount => _outputsCount);
                IF _inputsCount <> UINT#8 OR _outputsCount <> UINT#0 THEN
                    Messenger.Activate(UINT#916,eAxoMessageCategory#Error);
                    Status.Error.Id := UINT#916;
                    RETURN;
                END_IF;
                //******************Slot 21*****************//
                _geoAddr.Slot   :=  UINT#21;
                _geoAddr.HardwareType := UINT#4; // (4-Module)
                _retval := ReadHardwareIDFromSlot(geoAddr := _geoAddr, hardwareID => Config.HWIDs.HwID_out_1);
                IF Config.HWIDs.HwID_out_1 = UINT#0 THEN
                    Messenger.Activate(UINT#910,eAxoMessageCategory#Error);
                    Status.Error.Id := UINT#910;
                    RETURN;
                END_IF;
                IF _retval = WORD#8091 THEN
                    Messenger.Activate(UINT#911,eAxoMessageCategory#Error);
                    Status.Error.Id := UINT#911;
                    RETURN;
                END_IF;
                IF _retval = WORD#8094 THEN
                    Messenger.Activate(UINT#912,eAxoMessageCategory#Error);
                    Status.Error.Id := UINT#912;
                    RETURN;
                END_IF;
                IF _retval = WORD#8095 THEN
                    Messenger.Activate(UINT#913,eAxoMessageCategory#Error);
                    Status.Error.Id := UINT#913;
                    RETURN;
                END_IF;
                IF _retval = WORD#8096 THEN
                    Messenger.Activate(UINT#914,eAxoMessageCategory#Error);
                    Status.Error.Id := UINT#914;
                    RETURN;
                END_IF;
                IF _retval = WORD#8097 THEN
                    Messenger.Activate(UINT#715,eAxoMessageCategory#Error);
                    Status.Error.Id := UINT#715;
                    RETURN;
                END_IF;
                ReadHardwareIOAddress(hardwareID := (Config.HWIDs.HwID_out_1) , inputStartAddress => _inputsAddress , inputCount => _inputsCount , outputStartAddress => _outputsAddress , outputCount => _outputsCount);
                IF _outputsCount <> UINT#8 OR _inputsCount <> UINT#0 THEN
                    Messenger.Activate(UINT#916,eAxoMessageCategory#Error);
                    Status.Error.Id := UINT#916;
                    RETURN;
                END_IF;
                //******************Slot 22*****************//
                _geoAddr.Slot   :=  UINT#22;
                _geoAddr.HardwareType := UINT#4; // (4-Module)
                _retval := ReadHardwareIDFromSlot(geoAddr := _geoAddr, hardwareID => Config.HWIDs.HwID_out_2);
                IF Config.HWIDs.HwID_out_2 = UINT#0 THEN
                    Messenger.Activate(UINT#920,eAxoMessageCategory#Error);
                    Status.Error.Id := UINT#920;
                    RETURN;
                END_IF;
                IF _retval = WORD#8091 THEN
                    Messenger.Activate(UINT#921,eAxoMessageCategory#Error);
                    Status.Error.Id := UINT#921;
                    RETURN;
                END_IF;
                IF _retval = WORD#8094 THEN
                    Messenger.Activate(UINT#922,eAxoMessageCategory#Error);
                    Status.Error.Id := UINT#922;
                    RETURN;
                END_IF;
                IF _retval = WORD#8095 THEN
                    Messenger.Activate(UINT#923,eAxoMessageCategory#Error);
                    Status.Error.Id := UINT#923;
                    RETURN;
                END_IF;
                IF _retval = WORD#8096 THEN
                    Messenger.Activate(UINT#924,eAxoMessageCategory#Error);
                    Status.Error.Id := UINT#924;
                    RETURN;
                END_IF;
                IF _retval = WORD#8097 THEN
                    Messenger.Activate(UINT#925,eAxoMessageCategory#Error);
                    Status.Error.Id := UINT#925;
                    RETURN;
                END_IF;
                ReadHardwareIOAddress(hardwareID := (Config.HWIDs.HwID_out_2) , inputStartAddress => _inputsAddress , inputCount => _inputsCount , outputStartAddress => _outputsAddress , outputCount => _outputsCount);
                IF _outputsCount <> UINT#8 OR _inputsCount <> UINT#0 THEN
                    Messenger.Activate(UINT#926,eAxoMessageCategory#Error);
                    Status.Error.Id := UINT#926;
                    RETURN;
                END_IF;
                //******************Slot 23*****************//
                _geoAddr.Slot   :=  UINT#23;
                _geoAddr.HardwareType := UINT#4; // (4-Module)
                _retval := ReadHardwareIDFromSlot(geoAddr := _geoAddr, hardwareID => Config.HWIDs.HwID_out_3);
                IF Config.HWIDs.HwID_out_3 = UINT#0 THEN
                    Messenger.Activate(UINT#930,eAxoMessageCategory#Error);
                    Status.Error.Id := UINT#930;
                    RETURN;
                END_IF;
                IF _retval = WORD#8091 THEN
                    Messenger.Activate(UINT#931,eAxoMessageCategory#Error);
                    Status.Error.Id := UINT#931;
                    RETURN;
                END_IF;
                IF _retval = WORD#8094 THEN
                    Messenger.Activate(UINT#932,eAxoMessageCategory#Error);
                    Status.Error.Id := UINT#932;
                    RETURN;
                END_IF;
                IF _retval = WORD#8095 THEN
                    Messenger.Activate(UINT#933,eAxoMessageCategory#Error);
                    Status.Error.Id := UINT#933;
                    RETURN;
                END_IF;
                IF _retval = WORD#8096 THEN
                    Messenger.Activate(UINT#934,eAxoMessageCategory#Error);
                    Status.Error.Id := UINT#934;
                    RETURN;
                END_IF;
                IF _retval = WORD#8097 THEN
                    Messenger.Activate(UINT#935,eAxoMessageCategory#Error);
                    Status.Error.Id := UINT#935;
                    RETURN;
                END_IF;
                ReadHardwareIOAddress(hardwareID := (Config.HWIDs.HwID_out_3) , inputStartAddress => _inputsAddress , inputCount => _inputsCount , outputStartAddress => _outputsAddress , outputCount => _outputsCount);
                IF _outputsCount <> UINT#8 OR _inputsCount <> UINT#0 THEN
                    Messenger.Activate(UINT#936,eAxoMessageCategory#Error);
                    Status.Error.Id := UINT#936;
                    RETURN;
                END_IF;
                //******************Slot 24*****************//
                _geoAddr.Slot   :=  UINT#24;
                _geoAddr.HardwareType := UINT#4; // (4-Module)
                _retval := ReadHardwareIDFromSlot(geoAddr := _geoAddr, hardwareID => Config.HWIDs.HwID_out_4);
                IF Config.HWIDs.HwID_out_4 = UINT#0 THEN
                    Messenger.Activate(UINT#940,eAxoMessageCategory#Error);
                    Status.Error.Id := UINT#940;
                    RETURN;
                END_IF;
                IF _retval = WORD#8091 THEN
                    Messenger.Activate(UINT#941,eAxoMessageCategory#Error);
                    Status.Error.Id := UINT#941;
                    RETURN;
                END_IF;
                IF _retval = WORD#8094 THEN
                    Messenger.Activate(UINT#942,eAxoMessageCategory#Error);
                    Status.Error.Id := UINT#942;
                    RETURN;
                END_IF;
                IF _retval = WORD#8095 THEN
                    Messenger.Activate(UINT#943,eAxoMessageCategory#Error);
                    Status.Error.Id := UINT#943;
                    RETURN;
                END_IF;
                IF _retval = WORD#8096 THEN
                    Messenger.Activate(UINT#944,eAxoMessageCategory#Error);
                    Status.Error.Id := UINT#944;
                    RETURN;
                END_IF;
                IF _retval = WORD#8097 THEN
                    Messenger.Activate(UINT#945,eAxoMessageCategory#Error);
                    Status.Error.Id := UINT#945;
                    RETURN;
                END_IF;
                ReadHardwareIOAddress(hardwareID := (Config.HWIDs.HwID_out_4) , inputStartAddress => _inputsAddress , inputCount => _inputsCount , outputStartAddress => _outputsAddress , outputCount => _outputsCount);
                IF _outputsCount <> UINT#8 OR _inputsCount <> UINT#0 THEN
                    Messenger.Activate(UINT#946,eAxoMessageCategory#Error);
                    Status.Error.Id := UINT#946;
                    RETURN;
                END_IF;
                //******************Slot 25*****************//
                _geoAddr.Slot   :=  UINT#25;
                _geoAddr.HardwareType := UINT#4; // (4-Module)
                _retval := ReadHardwareIDFromSlot(geoAddr := _geoAddr, hardwareID => Config.HWIDs.HwID_out_5);
                IF Config.HWIDs.HwID_out_5 = UINT#0 THEN
                    Messenger.Activate(UINT#950,eAxoMessageCategory#Error);
                    Status.Error.Id := UINT#950;
                    RETURN;
                END_IF;
                IF _retval = WORD#8091 THEN
                    Messenger.Activate(UINT#951,eAxoMessageCategory#Error);
                    Status.Error.Id := UINT#951;
                    RETURN;
                END_IF;
                IF _retval = WORD#8094 THEN
                    Messenger.Activate(UINT#952,eAxoMessageCategory#Error);
                    Status.Error.Id := UINT#952;
                    RETURN;
                END_IF;
                IF _retval = WORD#8095 THEN
                    Messenger.Activate(UINT#953,eAxoMessageCategory#Error);
                    Status.Error.Id := UINT#953;
                    RETURN;
                END_IF;
                IF _retval = WORD#8096 THEN
                    Messenger.Activate(UINT#954,eAxoMessageCategory#Error);
                    Status.Error.Id := UINT#954;
                    RETURN;
                END_IF;
                IF _retval = WORD#8097 THEN
                    Messenger.Activate(UINT#955,eAxoMessageCategory#Error);
                    Status.Error.Id := UINT#955;
                    RETURN;
                END_IF;
                ReadHardwareIOAddress(hardwareID := (Config.HWIDs.HwID_out_5) , inputStartAddress => _inputsAddress , inputCount => _inputsCount , outputStartAddress => _outputsAddress , outputCount => _outputsCount);
                IF _outputsCount <> UINT#8 OR _inputsCount <> UINT#0 THEN
                    Messenger.Activate(UINT#956,eAxoMessageCategory#Error);
                    Status.Error.Id := UINT#956;
                    RETURN;
                END_IF;
                //******************Slot 26*****************//
                _geoAddr.Slot   :=  UINT#26;
                _geoAddr.HardwareType := UINT#4; // (4-Module)
                _retval := ReadHardwareIDFromSlot(geoAddr := _geoAddr, hardwareID => Config.HWIDs.HwID_out_6);
                IF Config.HWIDs.HwID_out_6 = UINT#0 THEN
                    Messenger.Activate(UINT#960,eAxoMessageCategory#Error);
                    Status.Error.Id := UINT#960;
                    RETURN;
                END_IF;
                IF _retval = WORD#8091 THEN
                    Messenger.Activate(UINT#961,eAxoMessageCategory#Error);
                    Status.Error.Id := UINT#961;
                    RETURN;
                END_IF;
                IF _retval = WORD#8094 THEN
                    Messenger.Activate(UINT#962,eAxoMessageCategory#Error);
                    Status.Error.Id := UINT#962;
                    RETURN;
                END_IF;
                IF _retval = WORD#8095 THEN
                    Messenger.Activate(UINT#963,eAxoMessageCategory#Error);
                    Status.Error.Id := UINT#963;
                    RETURN;
                END_IF;
                IF _retval = WORD#8096 THEN
                    Messenger.Activate(UINT#964,eAxoMessageCategory#Error);
                    Status.Error.Id := UINT#964;
                    RETURN;
                END_IF;
                IF _retval = WORD#8097 THEN
                    Messenger.Activate(UINT#965,eAxoMessageCategory#Error);
                    Status.Error.Id := UINT#965;
                    RETURN;
                END_IF;
                ReadHardwareIOAddress(hardwareID := (Config.HWIDs.HwID_out_6) , inputStartAddress => _inputsAddress , inputCount => _inputsCount , outputStartAddress => _outputsAddress , outputCount => _outputsCount);
                IF _outputsCount <> UINT#8 OR _inputsCount <> UINT#0 THEN
                    Messenger.Activate(UINT#966,eAxoMessageCategory#Error);
                    Status.Error.Id := UINT#966;
                    RETURN;
                END_IF;
                //******************Slot 27*****************//
                _geoAddr.Slot   :=  UINT#27;
                _geoAddr.HardwareType := UINT#4; // (4-Module)
                _retval := ReadHardwareIDFromSlot(geoAddr := _geoAddr, hardwareID => Config.HWIDs.HwID_out_7);
                IF Config.HWIDs.HwID_out_7 = UINT#0 THEN
                    Messenger.Activate(UINT#970,eAxoMessageCategory#Error);
                    Status.Error.Id := UINT#970;
                    RETURN;
                END_IF;
                IF _retval = WORD#8091 THEN
                    Messenger.Activate(UINT#971,eAxoMessageCategory#Error);
                    Status.Error.Id := UINT#971;
                    RETURN;
                END_IF;
                IF _retval = WORD#8094 THEN
                    Messenger.Activate(UINT#972,eAxoMessageCategory#Error);
                    Status.Error.Id := UINT#972;
                    RETURN;
                END_IF;
                IF _retval = WORD#8095 THEN
                    Messenger.Activate(UINT#973,eAxoMessageCategory#Error);
                    Status.Error.Id := UINT#973;
                    RETURN;
                END_IF;
                IF _retval = WORD#8096 THEN
                    Messenger.Activate(UINT#974,eAxoMessageCategory#Error);
                    Status.Error.Id := UINT#974;
                    RETURN;
                END_IF;
                IF _retval = WORD#8097 THEN
                    Messenger.Activate(UINT#975,eAxoMessageCategory#Error);
                    Status.Error.Id := UINT#975;
                    RETURN;
                END_IF;
                ReadHardwareIOAddress(hardwareID := (Config.HWIDs.HwID_out_7) , inputStartAddress => _inputsAddress , inputCount => _inputsCount , outputStartAddress => _outputsAddress , outputCount => _outputsCount);
                IF _outputsCount <> UINT#8 OR _inputsCount <> UINT#0 THEN
                    Messenger.Activate(UINT#976,eAxoMessageCategory#Error);
                    Status.Error.Id := UINT#976;
                    RETURN;
                END_IF;
                //******************Slot 28*****************//
                _geoAddr.Slot   :=  UINT#28;
                _geoAddr.HardwareType := UINT#4; // (4-Module)
                _retval := ReadHardwareIDFromSlot(geoAddr := _geoAddr, hardwareID => Config.HWIDs.HwID_out_8);
                IF Config.HWIDs.HwID_out_8 = UINT#0 THEN
                    Messenger.Activate(UINT#980,eAxoMessageCategory#Error);
                    Status.Error.Id := UINT#980;
                    RETURN;
                END_IF;
                IF _retval = WORD#8091 THEN
                    Messenger.Activate(UINT#981,eAxoMessageCategory#Error);
                    Status.Error.Id := UINT#981;
                    RETURN;
                END_IF;
                IF _retval = WORD#8094 THEN
                    Messenger.Activate(UINT#982,eAxoMessageCategory#Error);
                    Status.Error.Id := UINT#982;
                    RETURN;
                END_IF;
                IF _retval = WORD#8095 THEN
                    Messenger.Activate(UINT#983,eAxoMessageCategory#Error);
                    Status.Error.Id := UINT#983;
                    RETURN;
                END_IF;
                IF _retval = WORD#8096 THEN
                    Messenger.Activate(UINT#984,eAxoMessageCategory#Error);
                    Status.Error.Id := UINT#984;
                    RETURN;
                END_IF;
                IF _retval = WORD#8097 THEN
                    Messenger.Activate(UINT#985,eAxoMessageCategory#Error);
                    Status.Error.Id := UINT#985;
                    RETURN;
                END_IF;
                ReadHardwareIOAddress(hardwareID := (Config.HWIDs.HwID_out_8) , inputStartAddress => _inputsAddress , inputCount => _inputsCount , outputStartAddress => _outputsAddress , outputCount => _outputsCount);
                IF _outputsCount <> UINT#8 OR _inputsCount <> UINT#0 THEN
                    Messenger.Activate(UINT#986,eAxoMessageCategory#Error);
                    Status.Error.Id := UINT#986;
                    RETURN;
                END_IF;
                //******************Slot 29*****************//
                _geoAddr.Slot   :=  UINT#29;
                _geoAddr.HardwareType := UINT#4; // (4-Module)
                _retval := ReadHardwareIDFromSlot(geoAddr := _geoAddr, hardwareID => Config.HWIDs.HwID_out_9);
                IF Config.HWIDs.HwID_out_9 = UINT#0 THEN
                    Messenger.Activate(UINT#990,eAxoMessageCategory#Error);
                    Status.Error.Id := UINT#990;
                    RETURN;
                END_IF;
                IF _retval = WORD#8091 THEN
                    Messenger.Activate(UINT#991,eAxoMessageCategory#Error);
                    Status.Error.Id := UINT#991;
                    RETURN;
                END_IF;
                IF _retval = WORD#8094 THEN
                    Messenger.Activate(UINT#992,eAxoMessageCategory#Error);
                    Status.Error.Id := UINT#992;
                    RETURN;
                END_IF;
                IF _retval = WORD#8095 THEN
                    Messenger.Activate(UINT#993,eAxoMessageCategory#Error);
                    Status.Error.Id := UINT#993;
                    RETURN;
                END_IF;
                IF _retval = WORD#8096 THEN
                    Messenger.Activate(UINT#994,eAxoMessageCategory#Error);
                    Status.Error.Id := UINT#994;
                    RETURN;
                END_IF;
                IF _retval = WORD#8097 THEN
                    Messenger.Activate(UINT#995,eAxoMessageCategory#Error);
                    Status.Error.Id := UINT#995;
                    RETURN;
                END_IF;
                ReadHardwareIOAddress(hardwareID := (Config.HWIDs.HwID_out_9) , inputStartAddress => _inputsAddress , inputCount => _inputsCount , outputStartAddress => _outputsAddress , outputCount => _outputsCount);
                IF _outputsCount <> UINT#8 OR _inputsCount <> UINT#0 THEN
                    Messenger.Activate(UINT#996,eAxoMessageCategory#Error);
                    Status.Error.Id := UINT#996;
                    RETURN;
                END_IF;
                //******************Slot 30*****************//
                _geoAddr.Slot   :=  UINT#30;
                _geoAddr.HardwareType := UINT#4; // (4-Module)
                _retval := ReadHardwareIDFromSlot(geoAddr := _geoAddr, hardwareID => Config.HWIDs.HwID_out_10);
                IF Config.HWIDs.HwID_out_10 = UINT#0 THEN
                    Messenger.Activate(UINT#1000,eAxoMessageCategory#Error);
                    Status.Error.Id := UINT#1000;
                    RETURN;
                END_IF;
                IF _retval = WORD#8091 THEN
                    Messenger.Activate(UINT#1001,eAxoMessageCategory#Error);
                    Status.Error.Id := UINT#1001;
                    RETURN;
                END_IF;
                IF _retval = WORD#8094 THEN
                    Messenger.Activate(UINT#1002,eAxoMessageCategory#Error);
                    Status.Error.Id := UINT#1002;
                    RETURN;
                END_IF;
                IF _retval = WORD#8095 THEN
                    Messenger.Activate(UINT#1003,eAxoMessageCategory#Error);
                    Status.Error.Id := UINT#1003;
                    RETURN;
                END_IF;
                IF _retval = WORD#8096 THEN
                    Messenger.Activate(UINT#1004,eAxoMessageCategory#Error);
                    Status.Error.Id := UINT#1004;
                    RETURN;
                END_IF;
                IF _retval = WORD#8097 THEN
                    Messenger.Activate(UINT#1005,eAxoMessageCategory#Error);
                    Status.Error.Id := UINT#1005;
                    RETURN;
                END_IF;
                ReadHardwareIOAddress(hardwareID := (Config.HWIDs.HwID_out_10) , inputStartAddress => _inputsAddress , inputCount => _inputsCount , outputStartAddress => _outputsAddress , outputCount => _outputsCount);
                IF _outputsCount <> UINT#8 OR _inputsCount <> UINT#0 THEN
                    Messenger.Activate(UINT#1006,eAxoMessageCategory#Error);
                    Status.Error.Id := UINT#1006;
                    RETURN;
                END_IF;
                //******************Slot 31*****************//
                _geoAddr.Slot   :=  UINT#31;
                _geoAddr.HardwareType := UINT#4; // (4-Module)
                _retval := ReadHardwareIDFromSlot(geoAddr := _geoAddr, hardwareID => Config.HWIDs.HwID_out_11);
                IF Config.HWIDs.HwID_out_11 = UINT#0 THEN
                    Messenger.Activate(UINT#1010,eAxoMessageCategory#Error);
                    Status.Error.Id := UINT#1010;
                    RETURN;
                END_IF;
                IF _retval = WORD#8091 THEN
                    Messenger.Activate(UINT#1011,eAxoMessageCategory#Error);
                    Status.Error.Id := UINT#1011;
                    RETURN;
                END_IF;
                IF _retval = WORD#8094 THEN
                    Messenger.Activate(UINT#1012,eAxoMessageCategory#Error);
                    Status.Error.Id := UINT#1012;
                    RETURN;
                END_IF;
                IF _retval = WORD#8095 THEN
                    Messenger.Activate(UINT#1013,eAxoMessageCategory#Error);
                    Status.Error.Id := UINT#1013;
                    RETURN;
                END_IF;
                IF _retval = WORD#8096 THEN
                    Messenger.Activate(UINT#1014,eAxoMessageCategory#Error);
                    Status.Error.Id := UINT#1014;
                    RETURN;
                END_IF;
                IF _retval = WORD#8097 THEN
                    Messenger.Activate(UINT#1015,eAxoMessageCategory#Error);
                    Status.Error.Id := UINT#1015;
                    RETURN;
                END_IF;
                ReadHardwareIOAddress(hardwareID := (Config.HWIDs.HwID_out_11) , inputStartAddress => _inputsAddress , inputCount => _inputsCount , outputStartAddress => _outputsAddress , outputCount => _outputsCount);
                IF _outputsCount <> UINT#8 OR _inputsCount <> UINT#0 THEN
                    Messenger.Activate(UINT#1016,eAxoMessageCategory#Error);
                    Status.Error.Id := UINT#1016;
                    RETURN;
                END_IF;
                //******************Slot 32*****************//
                _geoAddr.Slot   :=  UINT#32;
                _geoAddr.HardwareType := UINT#4; // (4-Module)
                _retval := ReadHardwareIDFromSlot(geoAddr := _geoAddr, hardwareID => Config.HWIDs.HwID_out_12);
                IF Config.HWIDs.HwID_out_12 = UINT#0 THEN
                    Messenger.Activate(UINT#1020,eAxoMessageCategory#Error);
                    Status.Error.Id := UINT#1020;
                    RETURN;
                END_IF;
                IF _retval = WORD#8091 THEN
                    Messenger.Activate(UINT#1021,eAxoMessageCategory#Error);
                    Status.Error.Id := UINT#1021;
                    RETURN;
                END_IF;
                IF _retval = WORD#8094 THEN
                    Messenger.Activate(UINT#1022,eAxoMessageCategory#Error);
                    Status.Error.Id := UINT#1022;
                    RETURN;
                END_IF;
                IF _retval = WORD#8095 THEN
                    Messenger.Activate(UINT#1023,eAxoMessageCategory#Error);
                    Status.Error.Id := UINT#1023;
                    RETURN;
                END_IF;
                IF _retval = WORD#8096 THEN
                    Messenger.Activate(UINT#1024,eAxoMessageCategory#Error);
                    Status.Error.Id := UINT#1024;
                    RETURN;
                END_IF;
                IF _retval = WORD#8097 THEN
                    Messenger.Activate(UINT#1025,eAxoMessageCategory#Error);
                    Status.Error.Id := UINT#1025;
                    RETURN;
                END_IF;
                ReadHardwareIOAddress(hardwareID := (Config.HWIDs.HwID_out_12) , inputStartAddress => _inputsAddress , inputCount => _inputsCount , outputStartAddress => _outputsAddress , outputCount => _outputsCount);
                IF _outputsCount <> UINT#8 OR _inputsCount <> UINT#0 THEN
                    Messenger.Activate(UINT#1026,eAxoMessageCategory#Error);
                    Status.Error.Id := UINT#1026;
                    RETURN;
                END_IF;
                //******************Slot 33*****************//
                _geoAddr.Slot   :=  UINT#33;
                _geoAddr.HardwareType := UINT#4; // (4-Module)
                _retval := ReadHardwareIDFromSlot(geoAddr := _geoAddr, hardwareID => Config.HWIDs.HwID_out_13);
                IF Config.HWIDs.HwID_out_13 = UINT#0 THEN
                    Messenger.Activate(UINT#1030,eAxoMessageCategory#Error);
                    Status.Error.Id := UINT#1030;
                    RETURN;
                END_IF;
                IF _retval = WORD#8091 THEN
                    Messenger.Activate(UINT#1031,eAxoMessageCategory#Error);
                    Status.Error.Id := UINT#1031;
                    RETURN;
                END_IF;
                IF _retval = WORD#8094 THEN
                    Messenger.Activate(UINT#1032,eAxoMessageCategory#Error);
                    Status.Error.Id := UINT#1032;
                    RETURN;
                END_IF;
                IF _retval = WORD#8095 THEN
                    Messenger.Activate(UINT#1033,eAxoMessageCategory#Error);
                    Status.Error.Id := UINT#1033;
                    RETURN;
                END_IF;
                IF _retval = WORD#8096 THEN
                    Messenger.Activate(UINT#1034,eAxoMessageCategory#Error);
                    Status.Error.Id := UINT#1034;
                    RETURN;
                END_IF;
                IF _retval = WORD#8097 THEN
                    Messenger.Activate(UINT#1035,eAxoMessageCategory#Error);
                    Status.Error.Id := UINT#1035;
                    RETURN;
                END_IF;
                ReadHardwareIOAddress(hardwareID := (Config.HWIDs.HwID_out_13) , inputStartAddress => _inputsAddress , inputCount => _inputsCount , outputStartAddress => _outputsAddress , outputCount => _outputsCount);
                IF _outputsCount <> UINT#8 OR _inputsCount <> UINT#0 THEN
                    Messenger.Activate(UINT#1036,eAxoMessageCategory#Error);
                    Status.Error.Id := UINT#1036;
                    RETURN;
                END_IF;
                //******************Slot 34*****************//
                _geoAddr.Slot   :=  UINT#34;
                _geoAddr.HardwareType := UINT#4; // (4-Module)
                _retval := ReadHardwareIDFromSlot(geoAddr := _geoAddr, hardwareID => Config.HWIDs.HwID_out_14);
                IF Config.HWIDs.HwID_out_14 = UINT#0 THEN
                    Messenger.Activate(UINT#1040,eAxoMessageCategory#Error);
                    Status.Error.Id := UINT#1040;
                    RETURN;
                END_IF;
                IF _retval = WORD#8091 THEN
                    Messenger.Activate(UINT#1041,eAxoMessageCategory#Error);
                    Status.Error.Id := UINT#1041;
                    RETURN;
                END_IF;
                IF _retval = WORD#8094 THEN
                    Messenger.Activate(UINT#1042,eAxoMessageCategory#Error);
                    Status.Error.Id := UINT#1042;
                    RETURN;
                END_IF;
                IF _retval = WORD#8095 THEN
                    Messenger.Activate(UINT#1043,eAxoMessageCategory#Error);
                    Status.Error.Id := UINT#1043;
                    RETURN;
                END_IF;
                IF _retval = WORD#8096 THEN
                    Messenger.Activate(UINT#1044,eAxoMessageCategory#Error);
                    Status.Error.Id := UINT#1044;
                    RETURN;
                END_IF;
                IF _retval = WORD#8097 THEN
                    Messenger.Activate(UINT#1045,eAxoMessageCategory#Error);
                    Status.Error.Id := UINT#1045;
                    RETURN;
                END_IF;
                ReadHardwareIOAddress(hardwareID := (Config.HWIDs.HwID_out_14) , inputStartAddress => _inputsAddress , inputCount => _inputsCount , outputStartAddress => _outputsAddress , outputCount => _outputsCount);
                IF _outputsCount <> UINT#8 OR _inputsCount <> UINT#0 THEN
                    Messenger.Activate(UINT#1046,eAxoMessageCategory#Error);
                    Status.Error.Id := UINT#1046;
                    RETURN;
                END_IF;
                //******************Slot 35*****************//
                _geoAddr.Slot   :=  UINT#35;
                _geoAddr.HardwareType := UINT#4; // (4-Module)
                _retval := ReadHardwareIDFromSlot(geoAddr := _geoAddr, hardwareID => Config.HWIDs.HwID_out_15);
                IF Config.HWIDs.HwID_out_15 = UINT#0 THEN
                    Messenger.Activate(UINT#1050,eAxoMessageCategory#Error);
                    Status.Error.Id := UINT#1050;
                    RETURN;
                END_IF;
                IF _retval = WORD#8091 THEN
                    Messenger.Activate(UINT#1051,eAxoMessageCategory#Error);
                    Status.Error.Id := UINT#1051;
                    RETURN;
                END_IF;
                IF _retval = WORD#8094 THEN
                    Messenger.Activate(UINT#1052,eAxoMessageCategory#Error);
                    Status.Error.Id := UINT#1052;
                    RETURN;
                END_IF;
                IF _retval = WORD#8095 THEN
                    Messenger.Activate(UINT#1053,eAxoMessageCategory#Error);
                    Status.Error.Id := UINT#1053;
                    RETURN;
                END_IF;
                IF _retval = WORD#8096 THEN
                    Messenger.Activate(UINT#1054,eAxoMessageCategory#Error);
                    Status.Error.Id := UINT#1054;
                    RETURN;
                END_IF;
                IF _retval = WORD#8097 THEN
                    Messenger.Activate(UINT#1055,eAxoMessageCategory#Error);
                    Status.Error.Id := UINT#1055;
                    RETURN;
                END_IF;
                ReadHardwareIOAddress(hardwareID := (Config.HWIDs.HwID_out_15) , inputStartAddress => _inputsAddress , inputCount => _inputsCount , outputStartAddress => _outputsAddress , outputCount => _outputsCount);
                IF _outputsCount <> UINT#8 OR _inputsCount <> UINT#0 THEN
                    Messenger.Activate(UINT#1056,eAxoMessageCategory#Error);
                    Status.Error.Id := UINT#1056;
                    RETURN;
                END_IF;
                //******************Slot 36*****************//
                _geoAddr.Slot   :=  UINT#36;
                _geoAddr.HardwareType := UINT#4; // (4-Module)
                _retval := ReadHardwareIDFromSlot(geoAddr := _geoAddr, hardwareID => Config.HWIDs.HwID_out_16);
                IF Config.HWIDs.HwID_out_16 = UINT#0 THEN
                    Messenger.Activate(UINT#1060,eAxoMessageCategory#Error);
                    Status.Error.Id := UINT#1060;
                    RETURN;
                END_IF;
                IF _retval = WORD#8091 THEN
                    Messenger.Activate(UINT#1061,eAxoMessageCategory#Error);
                    Status.Error.Id := UINT#1061;
                    RETURN;
                END_IF;
                IF _retval = WORD#8094 THEN
                    Messenger.Activate(UINT#1062,eAxoMessageCategory#Error);
                    Status.Error.Id := UINT#1062;
                    RETURN;
                END_IF;
                IF _retval = WORD#8095 THEN
                    Messenger.Activate(UINT#1063,eAxoMessageCategory#Error);
                    Status.Error.Id := UINT#1063;
                    RETURN;
                END_IF;
                IF _retval = WORD#8096 THEN
                    Messenger.Activate(UINT#1064,eAxoMessageCategory#Error);
                    Status.Error.Id := UINT#1064;
                    RETURN;
                END_IF;
                IF _retval = WORD#8097 THEN
                    Messenger.Activate(UINT#1065,eAxoMessageCategory#Error);
                    Status.Error.Id := UINT#1065;
                    RETURN;
                END_IF;
                ReadHardwareIOAddress(hardwareID := (Config.HWIDs.HwID_out_16) , inputStartAddress => _inputsAddress , inputCount => _inputsCount , outputStartAddress => _outputsAddress , outputCount => _outputsCount);
                IF _outputsCount <> UINT#8 OR _inputsCount <> UINT#0 THEN
                    Messenger.Activate(UINT#1066,eAxoMessageCategory#Error);
                    Status.Error.Id := UINT#1066;
                    RETURN;
                END_IF;
                //******************Slot 37*****************//
                _geoAddr.Slot   :=  UINT#37;
                _geoAddr.HardwareType := UINT#4; // (4-Module)
                _retval := ReadHardwareIDFromSlot(geoAddr := _geoAddr, hardwareID => Config.HWIDs.HwID_out_17);
                IF Config.HWIDs.HwID_out_17 = UINT#0 THEN
                    Messenger.Activate(UINT#1070,eAxoMessageCategory#Error);
                    Status.Error.Id := UINT#1070;
                    RETURN;
                END_IF;
                IF _retval = WORD#8091 THEN
                    Messenger.Activate(UINT#1071,eAxoMessageCategory#Error);
                    Status.Error.Id := UINT#1071;
                    RETURN;
                END_IF;
                IF _retval = WORD#8094 THEN
                    Messenger.Activate(UINT#1072,eAxoMessageCategory#Error);
                    Status.Error.Id := UINT#1072;
                    RETURN;
                END_IF;
                IF _retval = WORD#8095 THEN
                    Messenger.Activate(UINT#1073,eAxoMessageCategory#Error);
                    Status.Error.Id := UINT#1073;
                    RETURN;
                END_IF;
                IF _retval = WORD#8096 THEN
                    Messenger.Activate(UINT#1074,eAxoMessageCategory#Error);
                    Status.Error.Id := UINT#1074;
                    RETURN;
                END_IF;
                IF _retval = WORD#8097 THEN
                    Messenger.Activate(UINT#1075,eAxoMessageCategory#Error);
                    Status.Error.Id := UINT#1075;
                    RETURN;
                END_IF;
                ReadHardwareIOAddress(hardwareID := (Config.HWIDs.HwID_out_17) , inputStartAddress => _inputsAddress , inputCount => _inputsCount , outputStartAddress => _outputsAddress , outputCount => _outputsCount);
                IF _outputsCount <> UINT#8 OR _inputsCount <> UINT#0 THEN
                    Messenger.Activate(UINT#1076,eAxoMessageCategory#Error);
                    Status.Error.Id := UINT#1076;
                    RETURN;
                END_IF;
                //******************Slot 38*****************//
                _geoAddr.Slot   :=  UINT#38;
                _geoAddr.HardwareType := UINT#4; // (4-Module)
                _retval := ReadHardwareIDFromSlot(geoAddr := _geoAddr, hardwareID => Config.HWIDs.HwID_out_18);
                IF Config.HWIDs.HwID_out_18 = UINT#0 THEN
                    Messenger.Activate(UINT#1080,eAxoMessageCategory#Error);
                    Status.Error.Id := UINT#1080;
                    RETURN;
                END_IF;
                IF _retval = WORD#8091 THEN
                    Messenger.Activate(UINT#1081,eAxoMessageCategory#Error);
                    Status.Error.Id := UINT#1081;
                    RETURN;
                END_IF;
                IF _retval = WORD#8094 THEN
                    Messenger.Activate(UINT#1082,eAxoMessageCategory#Error);
                    Status.Error.Id := UINT#1082;
                    RETURN;
                END_IF;
                IF _retval = WORD#8095 THEN
                    Messenger.Activate(UINT#1083,eAxoMessageCategory#Error);
                    Status.Error.Id := UINT#1083;
                    RETURN;
                END_IF;
                IF _retval = WORD#8096 THEN
                    Messenger.Activate(UINT#1084,eAxoMessageCategory#Error);
                    Status.Error.Id := UINT#1084;
                    RETURN;
                END_IF;
                IF _retval = WORD#8097 THEN
                    Messenger.Activate(UINT#1085,eAxoMessageCategory#Error);
                    Status.Error.Id := UINT#1085;
                    RETURN;
                END_IF;
                ReadHardwareIOAddress(hardwareID := (Config.HWIDs.HwID_out_18) , inputStartAddress => _inputsAddress , inputCount => _inputsCount , outputStartAddress => _outputsAddress , outputCount => _outputsCount);
                IF _outputsCount <> UINT#8 OR _inputsCount <> UINT#0 THEN
                    Messenger.Activate(UINT#1086,eAxoMessageCategory#Error);
                    Status.Error.Id := UINT#1086;
                    RETURN;
                END_IF;
                //******************Slot 39*****************//
                _geoAddr.Slot   :=  UINT#39;
                _geoAddr.HardwareType := UINT#4; // (4-Module)
                _retval := ReadHardwareIDFromSlot(geoAddr := _geoAddr, hardwareID => Config.HWIDs.HwID_out_19);
                IF Config.HWIDs.HwID_out_19 = UINT#0 THEN
                    Messenger.Activate(UINT#1090,eAxoMessageCategory#Error);
                    Status.Error.Id := UINT#1090;
                    RETURN;
                END_IF;
                IF _retval = WORD#8091 THEN
                    Messenger.Activate(UINT#1091,eAxoMessageCategory#Error);
                    Status.Error.Id := UINT#1091;
                    RETURN;
                END_IF;
                IF _retval = WORD#8094 THEN
                    Messenger.Activate(UINT#1092,eAxoMessageCategory#Error);
                    Status.Error.Id := UINT#1092;
                    RETURN;
                END_IF;
                IF _retval = WORD#8095 THEN
                    Messenger.Activate(UINT#1093,eAxoMessageCategory#Error);
                    Status.Error.Id := UINT#1093;
                    RETURN;
                END_IF;
                IF _retval = WORD#8096 THEN
                    Messenger.Activate(UINT#1094,eAxoMessageCategory#Error);
                    Status.Error.Id := UINT#1094;
                    RETURN;
                END_IF;
                IF _retval = WORD#8097 THEN
                    Messenger.Activate(UINT#1095,eAxoMessageCategory#Error);
                    Status.Error.Id := UINT#1095;
                    RETURN;
                END_IF;
                ReadHardwareIOAddress(hardwareID := (Config.HWIDs.HwID_out_19) , inputStartAddress => _inputsAddress , inputCount => _inputsCount , outputStartAddress => _outputsAddress , outputCount => _outputsCount);
                IF _outputsCount <> UINT#8 OR _inputsCount <> UINT#0 THEN
                    Messenger.Activate(UINT#1096,eAxoMessageCategory#Error);
                    Status.Error.Id := UINT#1096;
                    RETURN;
                END_IF;
                //******************Slot 40*****************//
                _geoAddr.Slot   :=  UINT#40;
                _geoAddr.HardwareType := UINT#4; // (4-Module)
                _retval := ReadHardwareIDFromSlot(geoAddr := _geoAddr, hardwareID => Config.HWIDs.HwID_out_20);
                IF Config.HWIDs.HwID_out_20 = UINT#0 THEN
                    Messenger.Activate(UINT#1100,eAxoMessageCategory#Error);
                    Status.Error.Id := UINT#1100;
                    RETURN;
                END_IF;
                IF _retval = WORD#8091 THEN
                    Messenger.Activate(UINT#1101,eAxoMessageCategory#Error);
                    Status.Error.Id := UINT#1101;
                    RETURN;
                END_IF;
                IF _retval = WORD#8094 THEN
                    Messenger.Activate(UINT#1102,eAxoMessageCategory#Error);
                    Status.Error.Id := UINT#1102;
                    RETURN;
                END_IF;
                IF _retval = WORD#8095 THEN
                    Messenger.Activate(UINT#1103,eAxoMessageCategory#Error);
                    Status.Error.Id := UINT#1103;
                    RETURN;
                END_IF;
                IF _retval = WORD#8096 THEN
                    Messenger.Activate(UINT#1104,eAxoMessageCategory#Error);
                    Status.Error.Id := UINT#1104;
                    RETURN;
                END_IF;
                IF _retval = WORD#8097 THEN
                    Messenger.Activate(UINT#1105,eAxoMessageCategory#Error);
                    Status.Error.Id := UINT#1105;
                    RETURN;
                END_IF;
                ReadHardwareIOAddress(hardwareID := (Config.HWIDs.HwID_out_20) , inputStartAddress => _inputsAddress , inputCount => _inputsCount , outputStartAddress => _outputsAddress , outputCount => _outputsCount);
                IF _outputsCount <> UINT#8 OR _inputsCount <> UINT#0 THEN
                    Messenger.Activate(UINT#1106,eAxoMessageCategory#Error);
                    Status.Error.Id := UINT#1106;
                    RETURN;
                END_IF;

                IF inParent = NULL THEN
                    Messenger.Activate(UINT#1130,eAxoMessageCategory#Error);
                    Status.Error.Id := UINT#1130;
                    RETURN;
                END_IF;
                IF Config.HWIDs.HW_Device  = UINT#0 THEN
                    Messenger.Activate(UINT#1131,eAxoMessageCategory#Error);
                    Status.Error.Id := UINT#1131;
                    RETURN;
                END_IF;
                IF Config.HWIDs.HwID_in_1  = UINT#0 THEN
                    Messenger.Activate(UINT#1132,eAxoMessageCategory#Error);
                    Status.Error.Id := UINT#1132;
                    RETURN;
                END_IF;
                IF Config.HWIDs.HwID_in_2  = UINT#0 THEN
                    Messenger.Activate(UINT#1133,eAxoMessageCategory#Error);
                    Status.Error.Id := UINT#1133;
                    RETURN;
                END_IF;
                IF Config.HWIDs.HwID_in_3  = UINT#0 THEN
                    Messenger.Activate(UINT#1134,eAxoMessageCategory#Error);
                    Status.Error.Id := UINT#1134;
                    RETURN;
                END_IF;
                IF Config.HWIDs.HwID_in_4  = UINT#0 THEN
                    Messenger.Activate(UINT#1135,eAxoMessageCategory#Error);
                    Status.Error.Id := UINT#1135;
                    RETURN;
                END_IF;
                IF Config.HWIDs.HwID_in_5  = UINT#0 THEN
                    Messenger.Activate(UINT#1136,eAxoMessageCategory#Error);
                    Status.Error.Id := UINT#1136;
                    RETURN;
                END_IF;
                IF Config.HWIDs.HwID_in_6  = UINT#0 THEN
                    Messenger.Activate(UINT#1137,eAxoMessageCategory#Error);
                    Status.Error.Id := UINT#1137;
                    RETURN;
                END_IF;
                IF Config.HWIDs.HwID_in_7  = UINT#0 THEN
                    Messenger.Activate(UINT#1138,eAxoMessageCategory#Error);
                    Status.Error.Id := UINT#1138;
                    RETURN;
                END_IF;
                IF Config.HWIDs.HwID_in_8  = UINT#0 THEN
                    Messenger.Activate(UINT#1139,eAxoMessageCategory#Error);
                    Status.Error.Id := UINT#1139;
                    RETURN;
                END_IF;
                IF Config.HWIDs.HwID_in_9  = UINT#0 THEN
                    Messenger.Activate(UINT#1140,eAxoMessageCategory#Error);
                    Status.Error.Id := UINT#1140;
                    RETURN;
                END_IF;
                IF Config.HWIDs.HwID_in_10  = UINT#0 THEN
                    Messenger.Activate(UINT#1141,eAxoMessageCategory#Error);
                    Status.Error.Id := UINT#1141;
                    RETURN;
                END_IF;
                IF Config.HWIDs.HwID_in_11  = UINT#0 THEN
                    Messenger.Activate(UINT#1142,eAxoMessageCategory#Error);
                    Status.Error.Id := UINT#1142;
                    RETURN;
                END_IF;
                IF Config.HWIDs.HwID_in_12  = UINT#0 THEN
                    Messenger.Activate(UINT#1143,eAxoMessageCategory#Error);
                    Status.Error.Id := UINT#1143;
                    RETURN;
                END_IF;
                IF Config.HWIDs.HwID_in_13  = UINT#0 THEN
                    Messenger.Activate(UINT#1144,eAxoMessageCategory#Error);
                    Status.Error.Id := UINT#1144;
                    RETURN;
                END_IF;
                IF Config.HWIDs.HwID_in_14  = UINT#0 THEN
                    Messenger.Activate(UINT#1145,eAxoMessageCategory#Error);
                    Status.Error.Id := UINT#1145;
                    RETURN;
                END_IF;
                IF Config.HWIDs.HwID_in_15  = UINT#0 THEN
                    Messenger.Activate(UINT#1146,eAxoMessageCategory#Error);
                    Status.Error.Id := UINT#1146;
                    RETURN;
                END_IF;
                IF Config.HWIDs.HwID_in_16  = UINT#0 THEN
                    Messenger.Activate(UINT#1147,eAxoMessageCategory#Error);
                    Status.Error.Id := UINT#1147;
                    RETURN;
                END_IF;
                IF Config.HWIDs.HwID_in_17  = UINT#0 THEN
                    Messenger.Activate(UINT#1148,eAxoMessageCategory#Error);
                    Status.Error.Id := UINT#1148;
                    RETURN;
                END_IF;
                IF Config.HWIDs.HwID_in_18  = UINT#0 THEN
                    Messenger.Activate(UINT#1149,eAxoMessageCategory#Error);
                    Status.Error.Id := UINT#1149;
                    RETURN;
                END_IF;
                IF Config.HWIDs.HwID_in_19  = UINT#0 THEN
                    Messenger.Activate(UINT#1150,eAxoMessageCategory#Error);
                    Status.Error.Id := UINT#1150;
                    RETURN;
                END_IF;
                IF Config.HWIDs.HwID_in_20  = UINT#0 THEN
                    Messenger.Activate(UINT#1151,eAxoMessageCategory#Error);
                    Status.Error.Id := UINT#1151;
                    RETURN;
                END_IF;
